PROGRAM P4_01_Write
VAR
	fbDBWrite		:FB_PLCDBWriteEvt(sNetId:=CONST.AMS_NETID, tTimeout:=DEFAULT_ADS_TIMEOUT);

	tableColumns	:ARRAY [0..5] OF STRING(50) := ['DateTime', 'User', 'Event', 'Description', 'OldValue', 'NewValue'];



	
	fbRecipeGeneral				:ARRAY[0..9] OF FB_AuditTrail_Write;
	fbRecipeProduction			:ARRAY[0..49] OF FB_AuditTrail_Write;
	fbRecipeCleaning			:ARRAY[0..49] OF FB_AuditTrail_Write;
	fbBatchProduction			:ARRAY[0..49] OF FB_AuditTrail_Write;
	fbBatchCleaning				:ARRAY[0..49] OF FB_AuditTrail_Write;
	
	fbMachine					:ARRAY[0..49] OF FB_AuditTrail_Write;
	fbSP						:ARRAY[0..49] OF FB_AuditTrail_Write;
	stDBParam 					:ST_AuditTrail;	
	
	//Cmd
	bWrite						:BOOL;								 
	bRead						:BOOL;
	sCmd						:STRING[300];
	nRecords					:UDINT;
	bFilter						:BOOL;
END_VAR

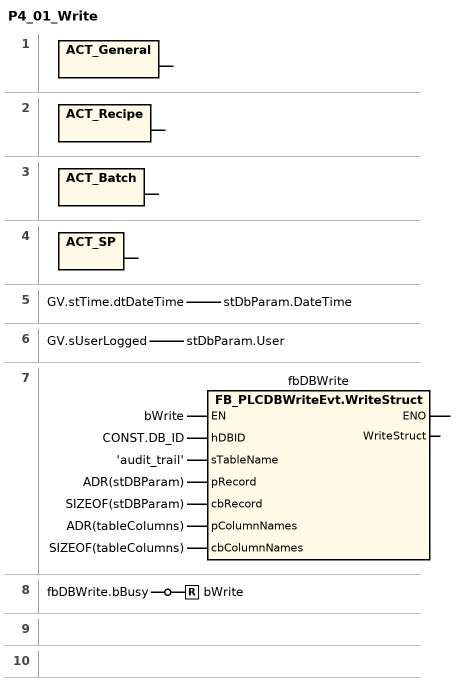
// NETWORK 1
ACT_General();

// NETWORK 2
ACT_Recipe();

// NETWORK 3
ACT_Batch();

// NETWORK 4
ACT_SP();

// NETWORK 5
stDbParam.DateTime := GV.stTime.dtDateTime;

// NETWORK 6
stDbParam.User := GV.sUserLogged;

// NETWORK 7
IF bWrite THEN
    fbDBWrite.WriteStruct(
        hDBID := CONST.DB_ID,
        sTableName := 'audit_trail',
        pRecord := ADR(stDBParam),
        cbRecord := SIZEOF(stDBParam),
        pColumnNames := ADR(tableColumns),
        cbColumnNames := SIZEOF(tableColumns));
END_IF

// NETWORK 8
bWrite R= NOT fbDBWrite.bBusy;

// NETWORK 9

// NETWORK 10

ACTION ACT_Batch:
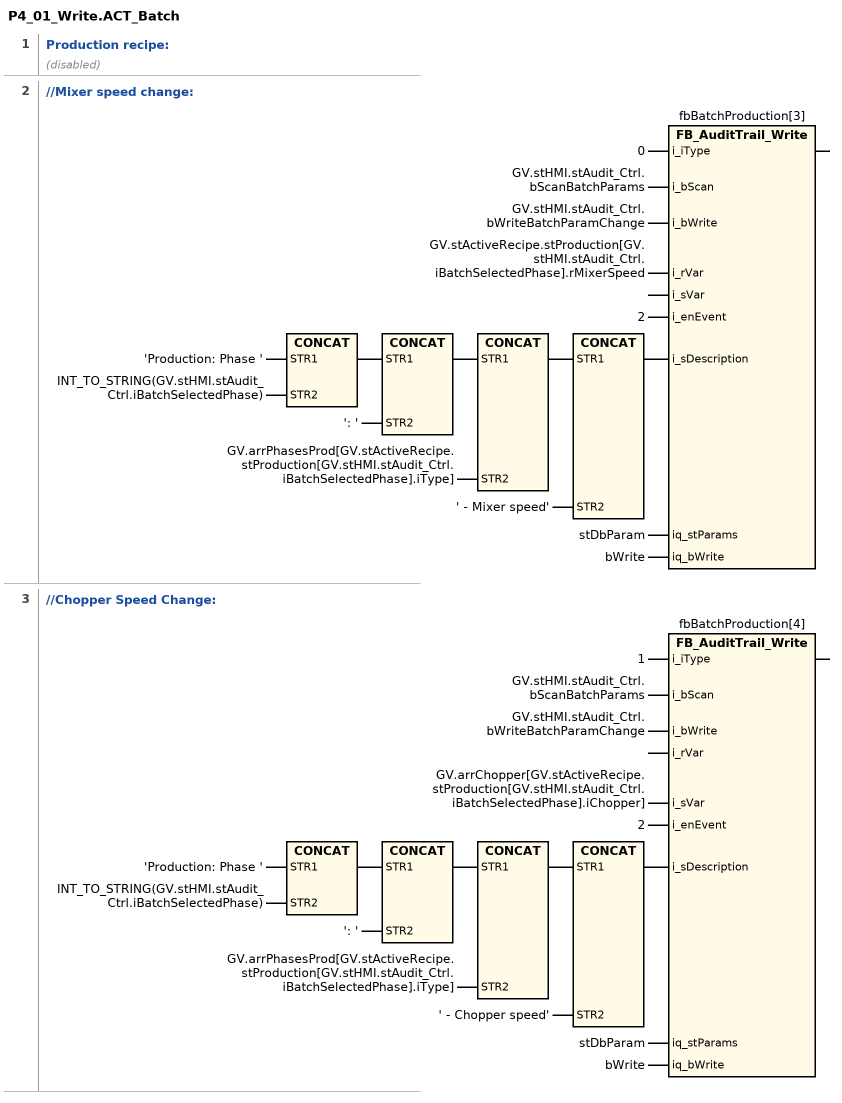
// NETWORK 1 (disabled)
// label: Production recipe

// NETWORK 2
// label: //Mixer speed change
fbBatchProduction[3](
    i_iType := 0,
    i_bScan := GV.stHMI.stAudit_Ctrl.bScanBatchParams,
    i_bWrite := GV.stHMI.stAudit_Ctrl.bWriteBatchParamChange,
    i_rVar := GV.stActiveRecipe.stProduction[GV.stHMI.stAudit_Ctrl.iBatchSelectedPhase].rMixerSpeed,
    i_enEvent := 2,
    i_sDescription := CONCAT(STR1 := CONCAT(STR1 := CONCAT(STR1 := CONCAT(STR1 := 'Production: Phase ', STR2 := INT_TO_STRING(GV.stHMI.stAudit_Ctrl.iBatchSelectedPhase)), STR2 := ': '), STR2 := GV.arrPhasesProd[GV.stActiveRecipe.stProduction[GV.stHMI.stAudit_Ctrl.iBatchSelectedPhase].iType]), STR2 := ' - Mixer speed'),
    iq_stParams := stDbParam,
    iq_bWrite := bWrite); // FB_AuditTrail_Write

// NETWORK 3
// label: //Chopper Speed Change
fbBatchProduction[4](
    i_iType := 1,
    i_bScan := GV.stHMI.stAudit_Ctrl.bScanBatchParams,
    i_bWrite := GV.stHMI.stAudit_Ctrl.bWriteBatchParamChange,
    i_sVar := GV.arrChopper[GV.stActiveRecipe.stProduction[GV.stHMI.stAudit_Ctrl.iBatchSelectedPhase].iChopper],
    i_enEvent := 2,
    i_sDescription := CONCAT(STR1 := CONCAT(STR1 := CONCAT(STR1 := CONCAT(STR1 := 'Production: Phase ', STR2 := INT_TO_STRING(GV.stHMI.stAudit_Ctrl.iBatchSelectedPhase)), STR2 := ': '), STR2 := GV.arrPhasesProd[GV.stActiveRecipe.stProduction[GV.stHMI.stAudit_Ctrl.iBatchSelectedPhase].iType]), STR2 := ' - Chopper speed'),
    iq_stParams := stDbParam,
    iq_bWrite := bWrite); // FB_AuditTrail_Write

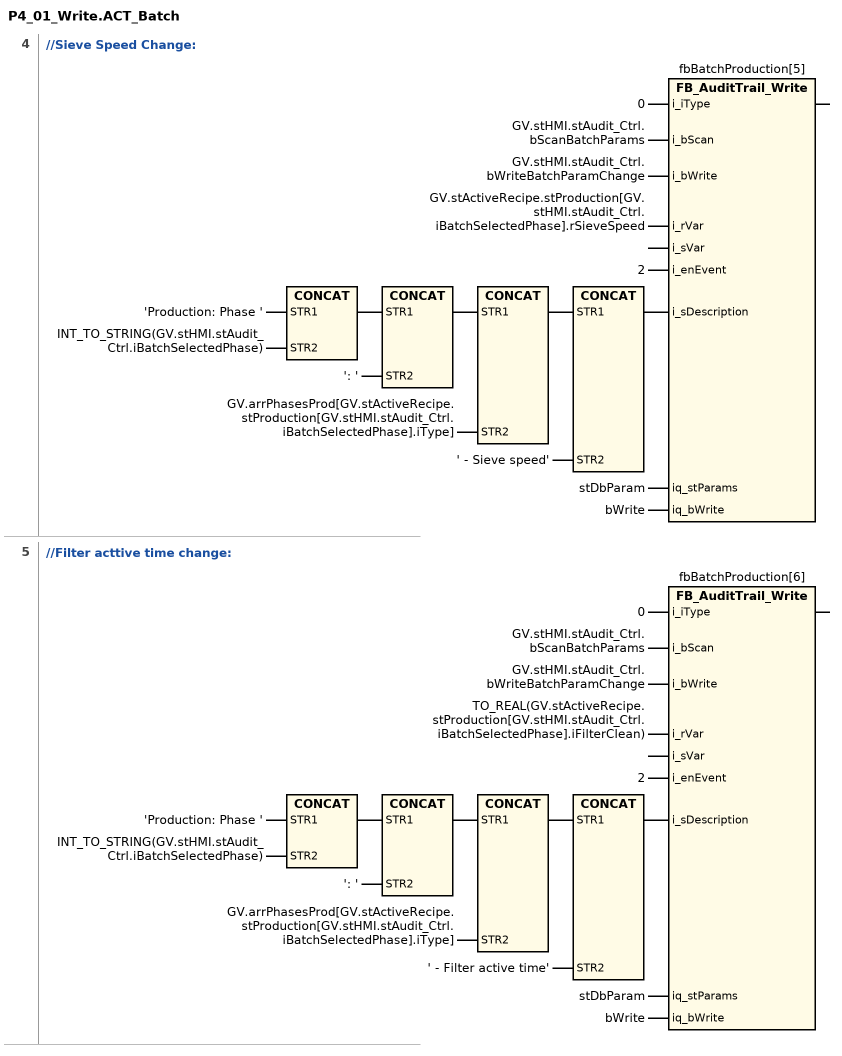
// NETWORK 4
// label: //Sieve Speed Change
fbBatchProduction[5](
    i_iType := 0,
    i_bScan := GV.stHMI.stAudit_Ctrl.bScanBatchParams,
    i_bWrite := GV.stHMI.stAudit_Ctrl.bWriteBatchParamChange,
    i_rVar := GV.stActiveRecipe.stProduction[GV.stHMI.stAudit_Ctrl.iBatchSelectedPhase].rSieveSpeed,
    i_enEvent := 2,
    i_sDescription := CONCAT(STR1 := CONCAT(STR1 := CONCAT(STR1 := CONCAT(STR1 := 'Production: Phase ', STR2 := INT_TO_STRING(GV.stHMI.stAudit_Ctrl.iBatchSelectedPhase)), STR2 := ': '), STR2 := GV.arrPhasesProd[GV.stActiveRecipe.stProduction[GV.stHMI.stAudit_Ctrl.iBatchSelectedPhase].iType]), STR2 := ' - Sieve speed'),
    iq_stParams := stDbParam,
    iq_bWrite := bWrite); // FB_AuditTrail_Write

// NETWORK 5
// label: //Filter acttive time change
fbBatchProduction[6](
    i_iType := 0,
    i_bScan := GV.stHMI.stAudit_Ctrl.bScanBatchParams,
    i_bWrite := GV.stHMI.stAudit_Ctrl.bWriteBatchParamChange,
    i_rVar := TO_REAL(GV.stActiveRecipe.stProduction[GV.stHMI.stAudit_Ctrl.iBatchSelectedPhase].iFilterClean),
    i_enEvent := 2,
    i_sDescription := CONCAT(STR1 := CONCAT(STR1 := CONCAT(STR1 := CONCAT(STR1 := 'Production: Phase ', STR2 := INT_TO_STRING(GV.stHMI.stAudit_Ctrl.iBatchSelectedPhase)), STR2 := ': '), STR2 := GV.arrPhasesProd[GV.stActiveRecipe.stProduction[GV.stHMI.stAudit_Ctrl.iBatchSelectedPhase].iType]), STR2 := ' - Filter active time'),
    iq_stParams := stDbParam,
    iq_bWrite := bWrite); // FB_AuditTrail_Write

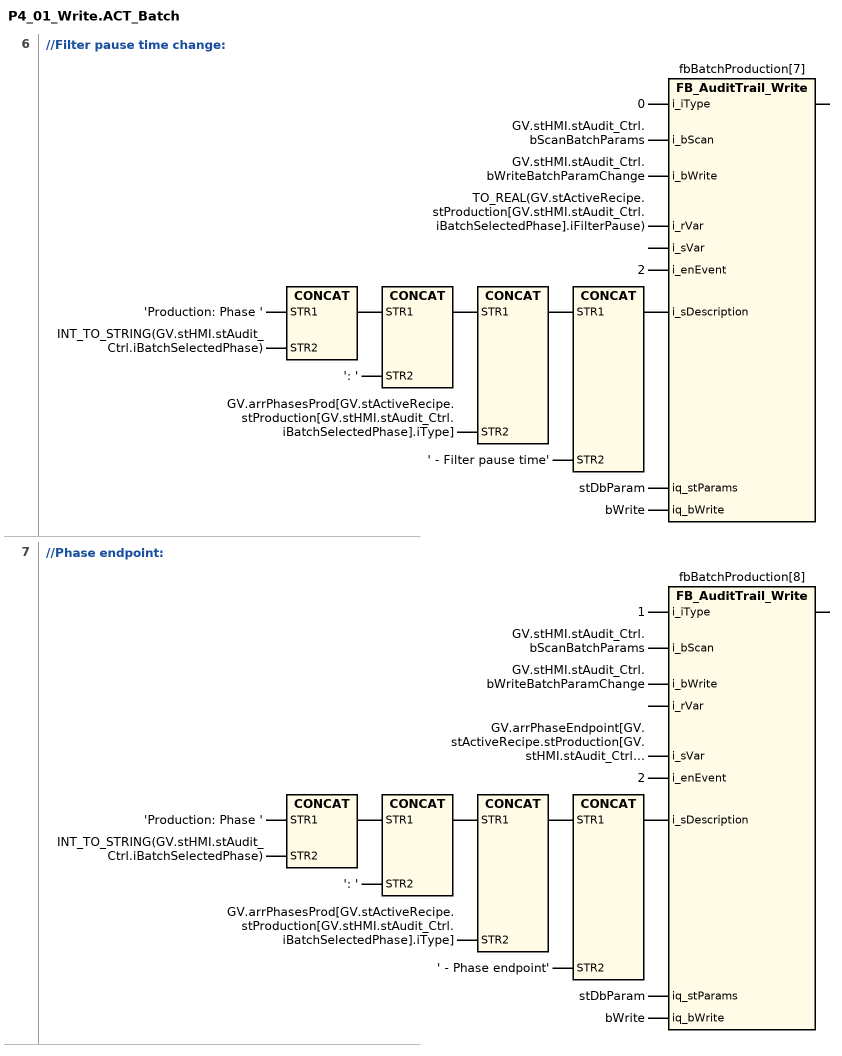
// NETWORK 6
// label: //Filter pause time change
fbBatchProduction[7](
    i_iType := 0,
    i_bScan := GV.stHMI.stAudit_Ctrl.bScanBatchParams,
    i_bWrite := GV.stHMI.stAudit_Ctrl.bWriteBatchParamChange,
    i_rVar := TO_REAL(GV.stActiveRecipe.stProduction[GV.stHMI.stAudit_Ctrl.iBatchSelectedPhase].iFilterPause),
    i_enEvent := 2,
    i_sDescription := CONCAT(STR1 := CONCAT(STR1 := CONCAT(STR1 := CONCAT(STR1 := 'Production: Phase ', STR2 := INT_TO_STRING(GV.stHMI.stAudit_Ctrl.iBatchSelectedPhase)), STR2 := ': '), STR2 := GV.arrPhasesProd[GV.stActiveRecipe.stProduction[GV.stHMI.stAudit_Ctrl.iBatchSelectedPhase].iType]), STR2 := ' - Filter pause time'),
    iq_stParams := stDbParam,
    iq_bWrite := bWrite); // FB_AuditTrail_Write

// NETWORK 7
// label: //Phase endpoint
fbBatchProduction[8](
    i_iType := 1,
    i_bScan := GV.stHMI.stAudit_Ctrl.bScanBatchParams,
    i_bWrite := GV.stHMI.stAudit_Ctrl.bWriteBatchParamChange,
    i_sVar := GV.arrPhaseEndpoint[GV.stActiveRecipe.stProduction[GV.stHMI.stAudit_Ctrl.iBatchSelectedPhase].iEndPoint],
    i_enEvent := 2,
    i_sDescription := CONCAT(STR1 := CONCAT(STR1 := CONCAT(STR1 := CONCAT(STR1 := 'Production: Phase ', STR2 := INT_TO_STRING(GV.stHMI.stAudit_Ctrl.iBatchSelectedPhase)), STR2 := ': '), STR2 := GV.arrPhasesProd[GV.stActiveRecipe.stProduction[GV.stHMI.stAudit_Ctrl.iBatchSelectedPhase].iType]), STR2 := ' - Phase endpoint'),
    iq_stParams := stDbParam,
    iq_bWrite := bWrite); // FB_AuditTrail_Write

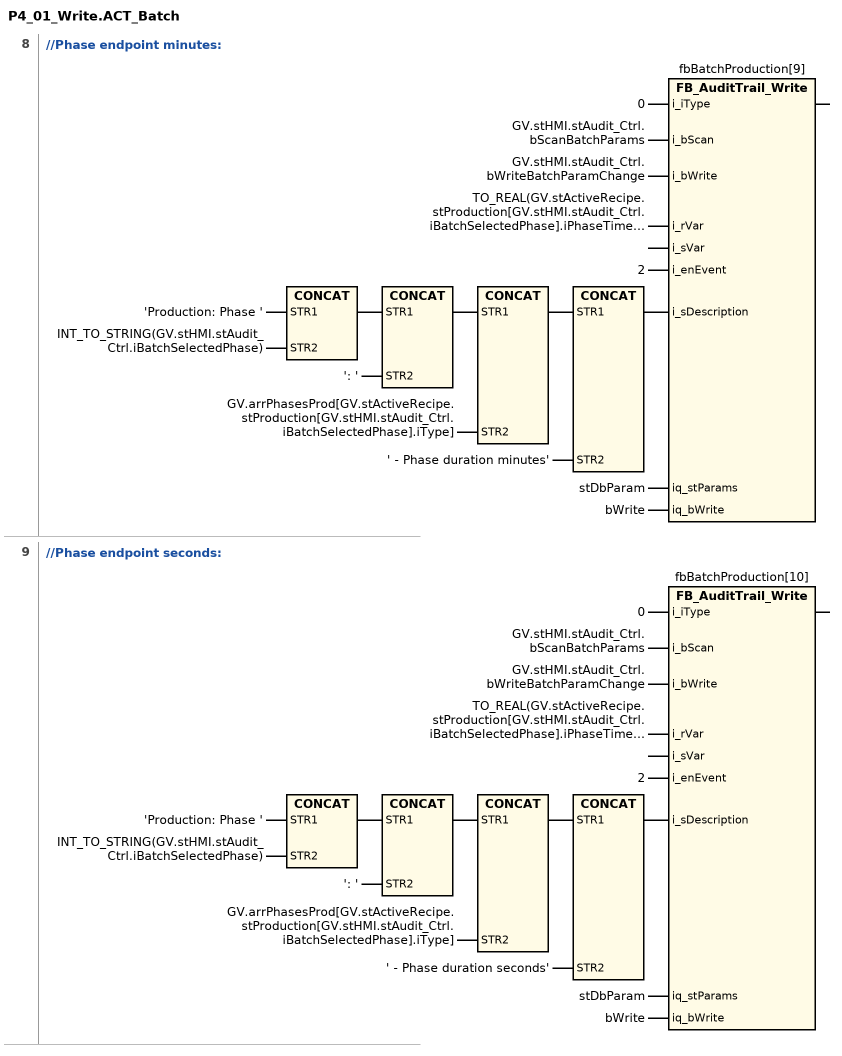
// NETWORK 8
// label: //Phase endpoint minutes
fbBatchProduction[9](
    i_iType := 0,
    i_bScan := GV.stHMI.stAudit_Ctrl.bScanBatchParams,
    i_bWrite := GV.stHMI.stAudit_Ctrl.bWriteBatchParamChange,
    i_rVar := TO_REAL(GV.stActiveRecipe.stProduction[GV.stHMI.stAudit_Ctrl.iBatchSelectedPhase].iPhaseTime.mins),
    i_enEvent := 2,
    i_sDescription := CONCAT(STR1 := CONCAT(STR1 := CONCAT(STR1 := CONCAT(STR1 := 'Production: Phase ', STR2 := INT_TO_STRING(GV.stHMI.stAudit_Ctrl.iBatchSelectedPhase)), STR2 := ': '), STR2 := GV.arrPhasesProd[GV.stActiveRecipe.stProduction[GV.stHMI.stAudit_Ctrl.iBatchSelectedPhase].iType]), STR2 := ' - Phase duration minutes'),
    iq_stParams := stDbParam,
    iq_bWrite := bWrite); // FB_AuditTrail_Write

// NETWORK 9
// label: //Phase endpoint seconds
fbBatchProduction[10](
    i_iType := 0,
    i_bScan := GV.stHMI.stAudit_Ctrl.bScanBatchParams,
    i_bWrite := GV.stHMI.stAudit_Ctrl.bWriteBatchParamChange,
    i_rVar := TO_REAL(GV.stActiveRecipe.stProduction[GV.stHMI.stAudit_Ctrl.iBatchSelectedPhase].iPhaseTime.sec),
    i_enEvent := 2,
    i_sDescription := CONCAT(STR1 := CONCAT(STR1 := CONCAT(STR1 := CONCAT(STR1 := 'Production: Phase ', STR2 := INT_TO_STRING(GV.stHMI.stAudit_Ctrl.iBatchSelectedPhase)), STR2 := ': '), STR2 := GV.arrPhasesProd[GV.stActiveRecipe.stProduction[GV.stHMI.stAudit_Ctrl.iBatchSelectedPhase].iType]), STR2 := ' - Phase duration seconds'),
    iq_stParams := stDbParam,
    iq_bWrite := bWrite); // FB_AuditTrail_Write

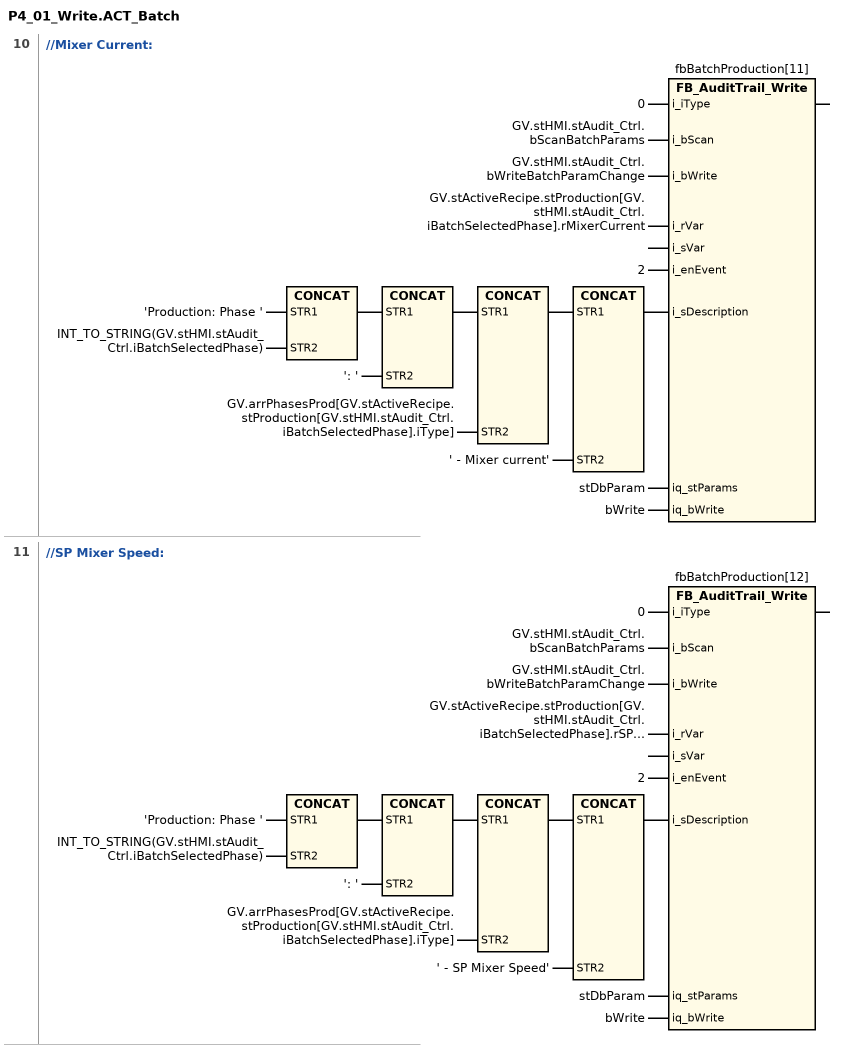
// NETWORK 10
// label: //Mixer Current
fbBatchProduction[11](
    i_iType := 0,
    i_bScan := GV.stHMI.stAudit_Ctrl.bScanBatchParams,
    i_bWrite := GV.stHMI.stAudit_Ctrl.bWriteBatchParamChange,
    i_rVar := GV.stActiveRecipe.stProduction[GV.stHMI.stAudit_Ctrl.iBatchSelectedPhase].rMixerCurrent,
    i_enEvent := 2,
    i_sDescription := CONCAT(STR1 := CONCAT(STR1 := CONCAT(STR1 := CONCAT(STR1 := 'Production: Phase ', STR2 := INT_TO_STRING(GV.stHMI.stAudit_Ctrl.iBatchSelectedPhase)), STR2 := ': '), STR2 := GV.arrPhasesProd[GV.stActiveRecipe.stProduction[GV.stHMI.stAudit_Ctrl.iBatchSelectedPhase].iType]), STR2 := ' - Mixer current'),
    iq_stParams := stDbParam,
    iq_bWrite := bWrite); // FB_AuditTrail_Write

// NETWORK 11
// label: //SP Mixer Speed
fbBatchProduction[12](
    i_iType := 0,
    i_bScan := GV.stHMI.stAudit_Ctrl.bScanBatchParams,
    i_bWrite := GV.stHMI.stAudit_Ctrl.bWriteBatchParamChange,
    i_rVar := GV.stActiveRecipe.stProduction[GV.stHMI.stAudit_Ctrl.iBatchSelectedPhase].rSP_MixingSpeed,
    i_enEvent := 2,
    i_sDescription := CONCAT(STR1 := CONCAT(STR1 := CONCAT(STR1 := CONCAT(STR1 := 'Production: Phase ', STR2 := INT_TO_STRING(GV.stHMI.stAudit_Ctrl.iBatchSelectedPhase)), STR2 := ': '), STR2 := GV.arrPhasesProd[GV.stActiveRecipe.stProduction[GV.stHMI.stAudit_Ctrl.iBatchSelectedPhase].iType]), STR2 := ' - SP Mixer Speed'),
    iq_stParams := stDbParam,
    iq_bWrite := bWrite); // FB_AuditTrail_Write

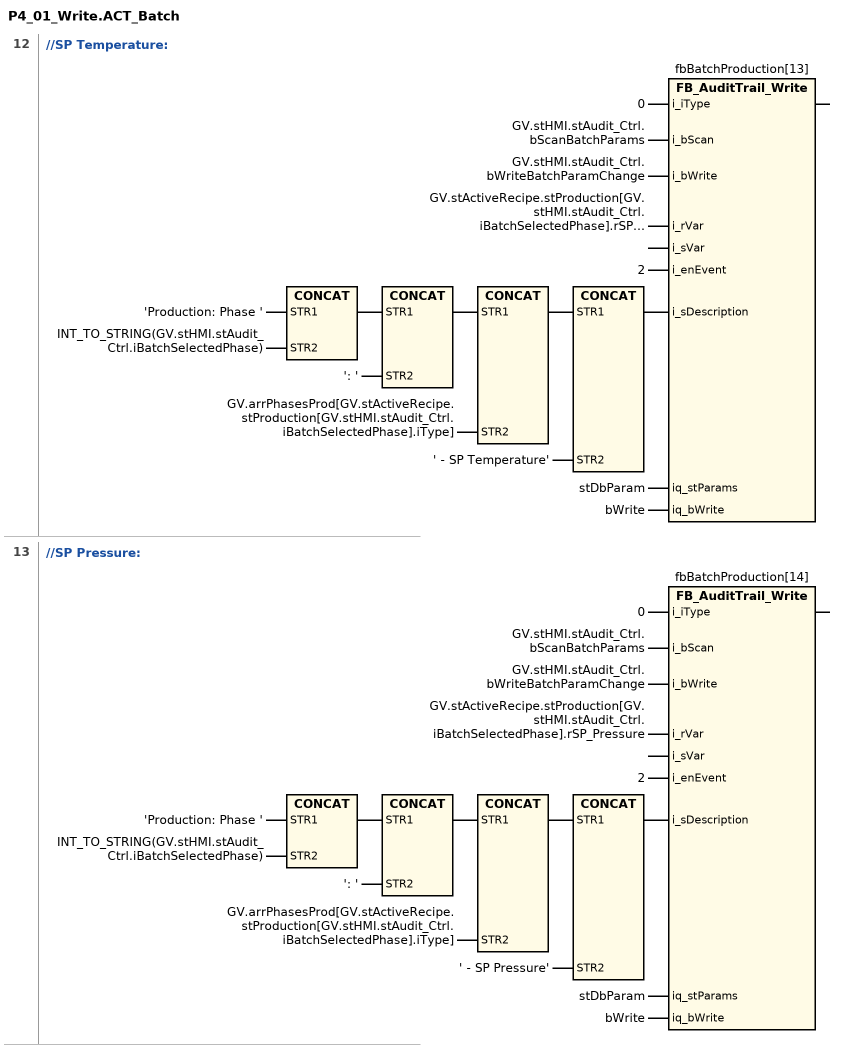
// NETWORK 12
// label: //SP Temperature
fbBatchProduction[13](
    i_iType := 0,
    i_bScan := GV.stHMI.stAudit_Ctrl.bScanBatchParams,
    i_bWrite := GV.stHMI.stAudit_Ctrl.bWriteBatchParamChange,
    i_rVar := GV.stActiveRecipe.stProduction[GV.stHMI.stAudit_Ctrl.iBatchSelectedPhase].rSP_Temperature,
    i_enEvent := 2,
    i_sDescription := CONCAT(STR1 := CONCAT(STR1 := CONCAT(STR1 := CONCAT(STR1 := 'Production: Phase ', STR2 := INT_TO_STRING(GV.stHMI.stAudit_Ctrl.iBatchSelectedPhase)), STR2 := ': '), STR2 := GV.arrPhasesProd[GV.stActiveRecipe.stProduction[GV.stHMI.stAudit_Ctrl.iBatchSelectedPhase].iType]), STR2 := ' - SP Temperature'),
    iq_stParams := stDbParam,
    iq_bWrite := bWrite); // FB_AuditTrail_Write

// NETWORK 13
// label: //SP Pressure
fbBatchProduction[14](
    i_iType := 0,
    i_bScan := GV.stHMI.stAudit_Ctrl.bScanBatchParams,
    i_bWrite := GV.stHMI.stAudit_Ctrl.bWriteBatchParamChange,
    i_rVar := GV.stActiveRecipe.stProduction[GV.stHMI.stAudit_Ctrl.iBatchSelectedPhase].rSP_Pressure,
    i_enEvent := 2,
    i_sDescription := CONCAT(STR1 := CONCAT(STR1 := CONCAT(STR1 := CONCAT(STR1 := 'Production: Phase ', STR2 := INT_TO_STRING(GV.stHMI.stAudit_Ctrl.iBatchSelectedPhase)), STR2 := ': '), STR2 := GV.arrPhasesProd[GV.stActiveRecipe.stProduction[GV.stHMI.stAudit_Ctrl.iBatchSelectedPhase].iType]), STR2 := ' - SP Pressure'),
    iq_stParams := stDbParam,
    iq_bWrite := bWrite); // FB_AuditTrail_Write

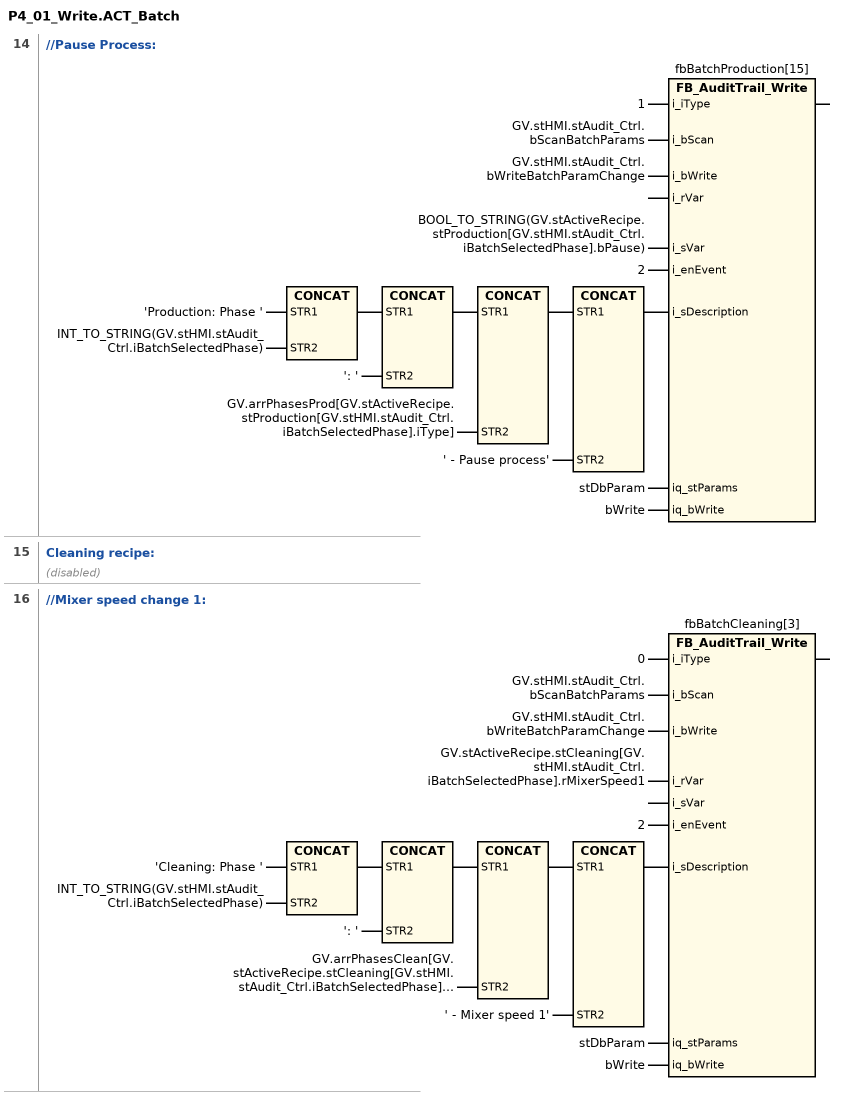
// NETWORK 14
// label: //Pause Process
fbBatchProduction[15](
    i_iType := 1,
    i_bScan := GV.stHMI.stAudit_Ctrl.bScanBatchParams,
    i_bWrite := GV.stHMI.stAudit_Ctrl.bWriteBatchParamChange,
    i_sVar := BOOL_TO_STRING(GV.stActiveRecipe.stProduction[GV.stHMI.stAudit_Ctrl.iBatchSelectedPhase].bPause),
    i_enEvent := 2,
    i_sDescription := CONCAT(STR1 := CONCAT(STR1 := CONCAT(STR1 := CONCAT(STR1 := 'Production: Phase ', STR2 := INT_TO_STRING(GV.stHMI.stAudit_Ctrl.iBatchSelectedPhase)), STR2 := ': '), STR2 := GV.arrPhasesProd[GV.stActiveRecipe.stProduction[GV.stHMI.stAudit_Ctrl.iBatchSelectedPhase].iType]), STR2 := ' - Pause process'),
    iq_stParams := stDbParam,
    iq_bWrite := bWrite); // FB_AuditTrail_Write

// NETWORK 15 (disabled)
// label: Cleaning recipe

// NETWORK 16
// label: //Mixer speed change 1
fbBatchCleaning[3](
    i_iType := 0,
    i_bScan := GV.stHMI.stAudit_Ctrl.bScanBatchParams,
    i_bWrite := GV.stHMI.stAudit_Ctrl.bWriteBatchParamChange,
    i_rVar := GV.stActiveRecipe.stCleaning[GV.stHMI.stAudit_Ctrl.iBatchSelectedPhase].rMixerSpeed1,
    i_enEvent := 2,
    i_sDescription := CONCAT(STR1 := CONCAT(STR1 := CONCAT(STR1 := CONCAT(STR1 := 'Cleaning: Phase ', STR2 := INT_TO_STRING(GV.stHMI.stAudit_Ctrl.iBatchSelectedPhase)), STR2 := ': '), STR2 := GV.arrPhasesClean[GV.stActiveRecipe.stCleaning[GV.stHMI.stAudit_Ctrl.iBatchSelectedPhase].iType]), STR2 := ' - Mixer speed 1'),
    iq_stParams := stDbParam,
    iq_bWrite := bWrite); // FB_AuditTrail_Write

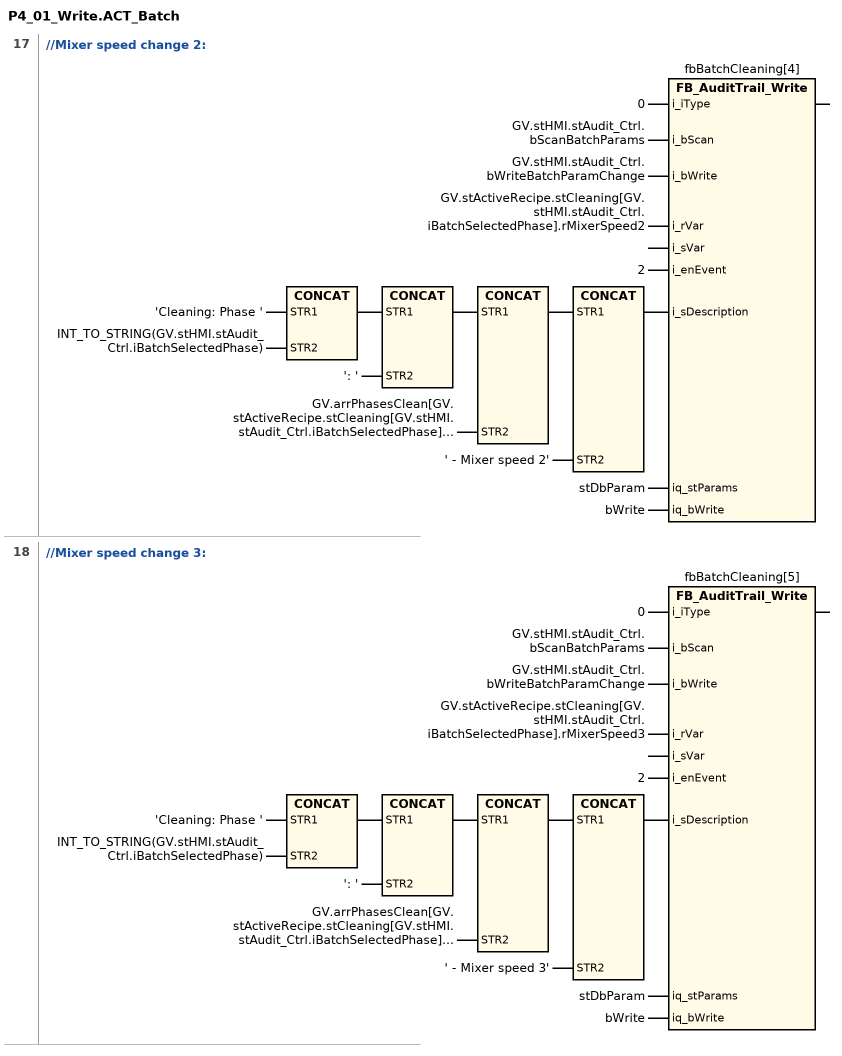
// NETWORK 17
// label: //Mixer speed change 2
fbBatchCleaning[4](
    i_iType := 0,
    i_bScan := GV.stHMI.stAudit_Ctrl.bScanBatchParams,
    i_bWrite := GV.stHMI.stAudit_Ctrl.bWriteBatchParamChange,
    i_rVar := GV.stActiveRecipe.stCleaning[GV.stHMI.stAudit_Ctrl.iBatchSelectedPhase].rMixerSpeed2,
    i_enEvent := 2,
    i_sDescription := CONCAT(STR1 := CONCAT(STR1 := CONCAT(STR1 := CONCAT(STR1 := 'Cleaning: Phase ', STR2 := INT_TO_STRING(GV.stHMI.stAudit_Ctrl.iBatchSelectedPhase)), STR2 := ': '), STR2 := GV.arrPhasesClean[GV.stActiveRecipe.stCleaning[GV.stHMI.stAudit_Ctrl.iBatchSelectedPhase].iType]), STR2 := ' - Mixer speed 2'),
    iq_stParams := stDbParam,
    iq_bWrite := bWrite); // FB_AuditTrail_Write

// NETWORK 18
// label: //Mixer speed change 3
fbBatchCleaning[5](
    i_iType := 0,
    i_bScan := GV.stHMI.stAudit_Ctrl.bScanBatchParams,
    i_bWrite := GV.stHMI.stAudit_Ctrl.bWriteBatchParamChange,
    i_rVar := GV.stActiveRecipe.stCleaning[GV.stHMI.stAudit_Ctrl.iBatchSelectedPhase].rMixerSpeed3,
    i_enEvent := 2,
    i_sDescription := CONCAT(STR1 := CONCAT(STR1 := CONCAT(STR1 := CONCAT(STR1 := 'Cleaning: Phase ', STR2 := INT_TO_STRING(GV.stHMI.stAudit_Ctrl.iBatchSelectedPhase)), STR2 := ': '), STR2 := GV.arrPhasesClean[GV.stActiveRecipe.stCleaning[GV.stHMI.stAudit_Ctrl.iBatchSelectedPhase].iType]), STR2 := ' - Mixer speed 3'),
    iq_stParams := stDbParam,
    iq_bWrite := bWrite); // FB_AuditTrail_Write

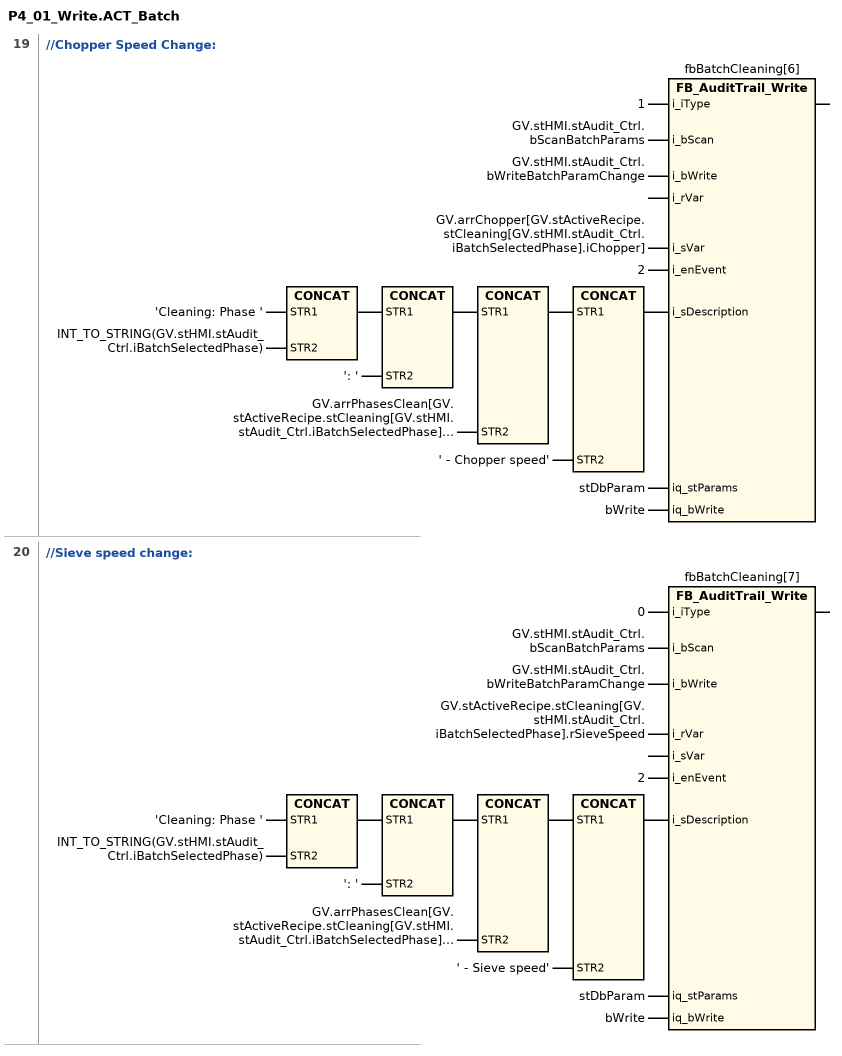
// NETWORK 19
// label: //Chopper Speed Change
fbBatchCleaning[6](
    i_iType := 1,
    i_bScan := GV.stHMI.stAudit_Ctrl.bScanBatchParams,
    i_bWrite := GV.stHMI.stAudit_Ctrl.bWriteBatchParamChange,
    i_sVar := GV.arrChopper[GV.stActiveRecipe.stCleaning[GV.stHMI.stAudit_Ctrl.iBatchSelectedPhase].iChopper],
    i_enEvent := 2,
    i_sDescription := CONCAT(STR1 := CONCAT(STR1 := CONCAT(STR1 := CONCAT(STR1 := 'Cleaning: Phase ', STR2 := INT_TO_STRING(GV.stHMI.stAudit_Ctrl.iBatchSelectedPhase)), STR2 := ': '), STR2 := GV.arrPhasesClean[GV.stActiveRecipe.stCleaning[GV.stHMI.stAudit_Ctrl.iBatchSelectedPhase].iType]), STR2 := ' - Chopper speed'),
    iq_stParams := stDbParam,
    iq_bWrite := bWrite); // FB_AuditTrail_Write

// NETWORK 20
// label: //Sieve speed change
fbBatchCleaning[7](
    i_iType := 0,
    i_bScan := GV.stHMI.stAudit_Ctrl.bScanBatchParams,
    i_bWrite := GV.stHMI.stAudit_Ctrl.bWriteBatchParamChange,
    i_rVar := GV.stActiveRecipe.stCleaning[GV.stHMI.stAudit_Ctrl.iBatchSelectedPhase].rSieveSpeed,
    i_enEvent := 2,
    i_sDescription := CONCAT(STR1 := CONCAT(STR1 := CONCAT(STR1 := CONCAT(STR1 := 'Cleaning: Phase ', STR2 := INT_TO_STRING(GV.stHMI.stAudit_Ctrl.iBatchSelectedPhase)), STR2 := ': '), STR2 := GV.arrPhasesClean[GV.stActiveRecipe.stCleaning[GV.stHMI.stAudit_Ctrl.iBatchSelectedPhase].iType]), STR2 := ' - Sieve speed'),
    iq_stParams := stDbParam,
    iq_bWrite := bWrite); // FB_AuditTrail_Write

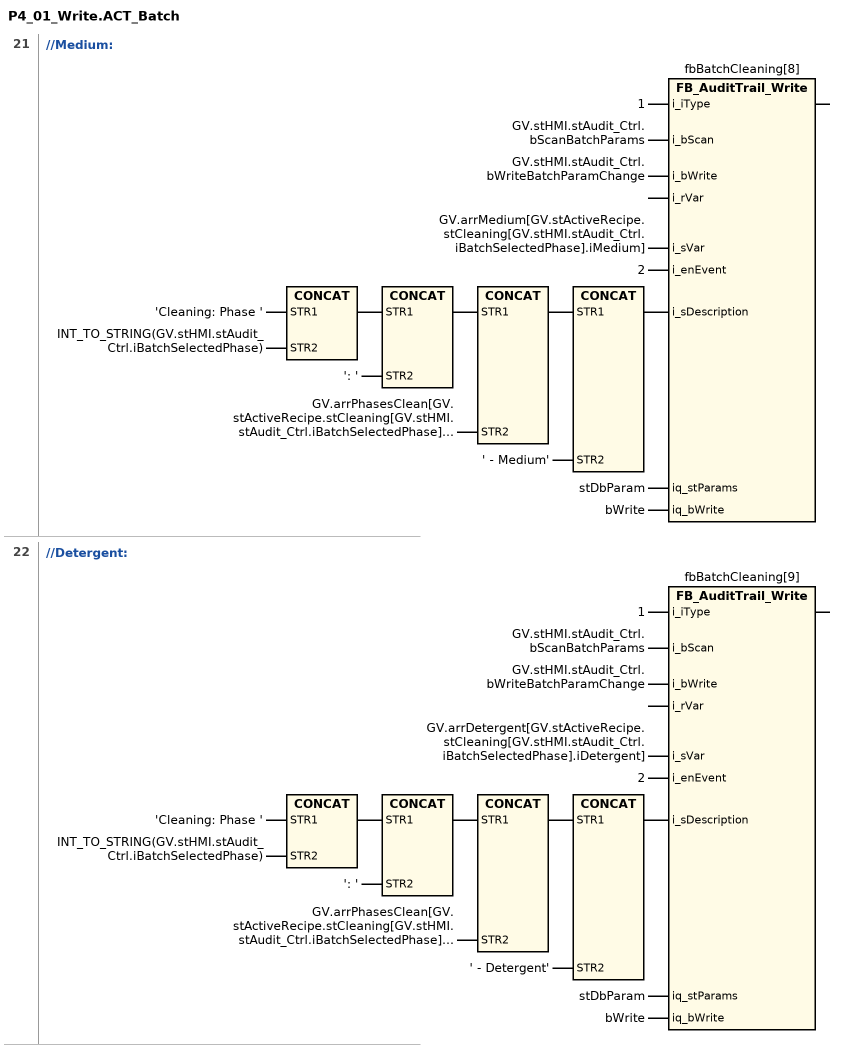
// NETWORK 21
// label: //Medium
fbBatchCleaning[8](
    i_iType := 1,
    i_bScan := GV.stHMI.stAudit_Ctrl.bScanBatchParams,
    i_bWrite := GV.stHMI.stAudit_Ctrl.bWriteBatchParamChange,
    i_sVar := GV.arrMedium[GV.stActiveRecipe.stCleaning[GV.stHMI.stAudit_Ctrl.iBatchSelectedPhase].iMedium],
    i_enEvent := 2,
    i_sDescription := CONCAT(STR1 := CONCAT(STR1 := CONCAT(STR1 := CONCAT(STR1 := 'Cleaning: Phase ', STR2 := INT_TO_STRING(GV.stHMI.stAudit_Ctrl.iBatchSelectedPhase)), STR2 := ': '), STR2 := GV.arrPhasesClean[GV.stActiveRecipe.stCleaning[GV.stHMI.stAudit_Ctrl.iBatchSelectedPhase].iType]), STR2 := ' - Medium'),
    iq_stParams := stDbParam,
    iq_bWrite := bWrite); // FB_AuditTrail_Write

// NETWORK 22
// label: //Detergent
fbBatchCleaning[9](
    i_iType := 1,
    i_bScan := GV.stHMI.stAudit_Ctrl.bScanBatchParams,
    i_bWrite := GV.stHMI.stAudit_Ctrl.bWriteBatchParamChange,
    i_sVar := GV.arrDetergent[GV.stActiveRecipe.stCleaning[GV.stHMI.stAudit_Ctrl.iBatchSelectedPhase].iDetergent],
    i_enEvent := 2,
    i_sDescription := CONCAT(STR1 := CONCAT(STR1 := CONCAT(STR1 := CONCAT(STR1 := 'Cleaning: Phase ', STR2 := INT_TO_STRING(GV.stHMI.stAudit_Ctrl.iBatchSelectedPhase)), STR2 := ': '), STR2 := GV.arrPhasesClean[GV.stActiveRecipe.stCleaning[GV.stHMI.stAudit_Ctrl.iBatchSelectedPhase].iType]), STR2 := ' - Detergent'),
    iq_stParams := stDbParam,
    iq_bWrite := bWrite); // FB_AuditTrail_Write

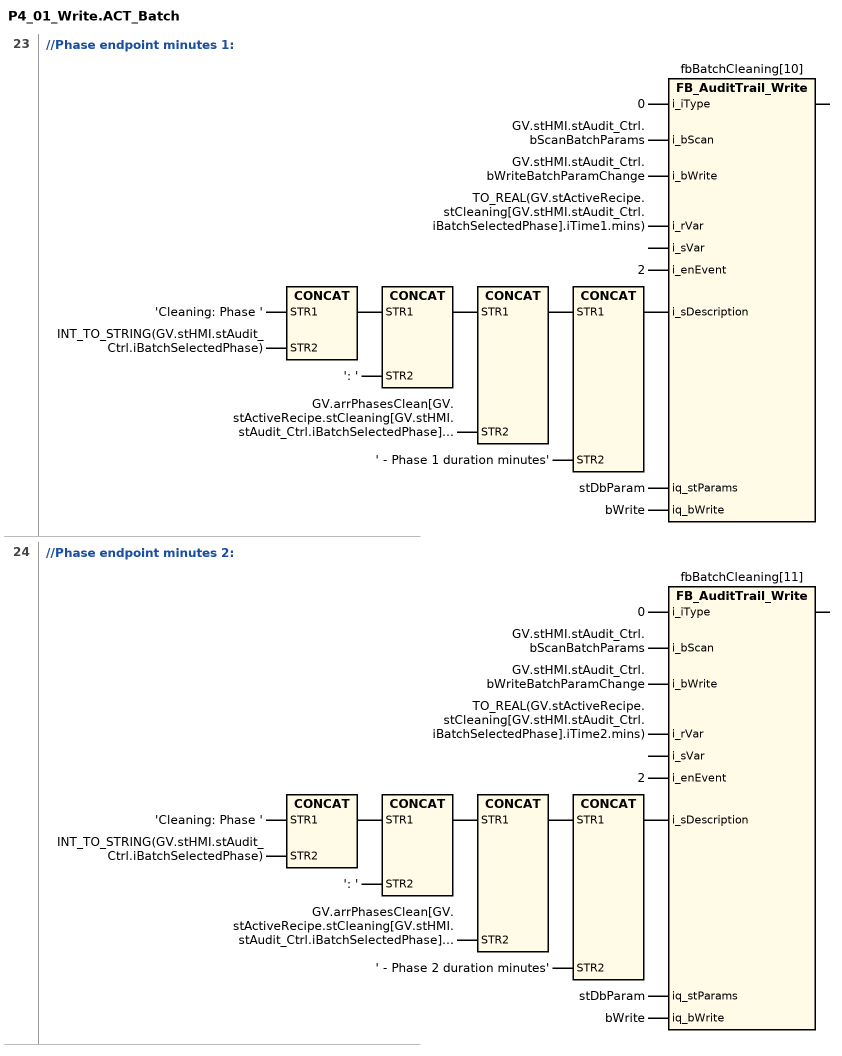
// NETWORK 23
// label: //Phase endpoint minutes 1
fbBatchCleaning[10](
    i_iType := 0,
    i_bScan := GV.stHMI.stAudit_Ctrl.bScanBatchParams,
    i_bWrite := GV.stHMI.stAudit_Ctrl.bWriteBatchParamChange,
    i_rVar := TO_REAL(GV.stActiveRecipe.stCleaning[GV.stHMI.stAudit_Ctrl.iBatchSelectedPhase].iTime1.mins),
    i_enEvent := 2,
    i_sDescription := CONCAT(STR1 := CONCAT(STR1 := CONCAT(STR1 := CONCAT(STR1 := 'Cleaning: Phase ', STR2 := INT_TO_STRING(GV.stHMI.stAudit_Ctrl.iBatchSelectedPhase)), STR2 := ': '), STR2 := GV.arrPhasesClean[GV.stActiveRecipe.stCleaning[GV.stHMI.stAudit_Ctrl.iBatchSelectedPhase].iType]), STR2 := ' - Phase 1 duration minutes'),
    iq_stParams := stDbParam,
    iq_bWrite := bWrite); // FB_AuditTrail_Write

// NETWORK 24
// label: //Phase endpoint minutes 2
fbBatchCleaning[11](
    i_iType := 0,
    i_bScan := GV.stHMI.stAudit_Ctrl.bScanBatchParams,
    i_bWrite := GV.stHMI.stAudit_Ctrl.bWriteBatchParamChange,
    i_rVar := TO_REAL(GV.stActiveRecipe.stCleaning[GV.stHMI.stAudit_Ctrl.iBatchSelectedPhase].iTime2.mins),
    i_enEvent := 2,
    i_sDescription := CONCAT(STR1 := CONCAT(STR1 := CONCAT(STR1 := CONCAT(STR1 := 'Cleaning: Phase ', STR2 := INT_TO_STRING(GV.stHMI.stAudit_Ctrl.iBatchSelectedPhase)), STR2 := ': '), STR2 := GV.arrPhasesClean[GV.stActiveRecipe.stCleaning[GV.stHMI.stAudit_Ctrl.iBatchSelectedPhase].iType]), STR2 := ' - Phase 2 duration minutes'),
    iq_stParams := stDbParam,
    iq_bWrite := bWrite); // FB_AuditTrail_Write

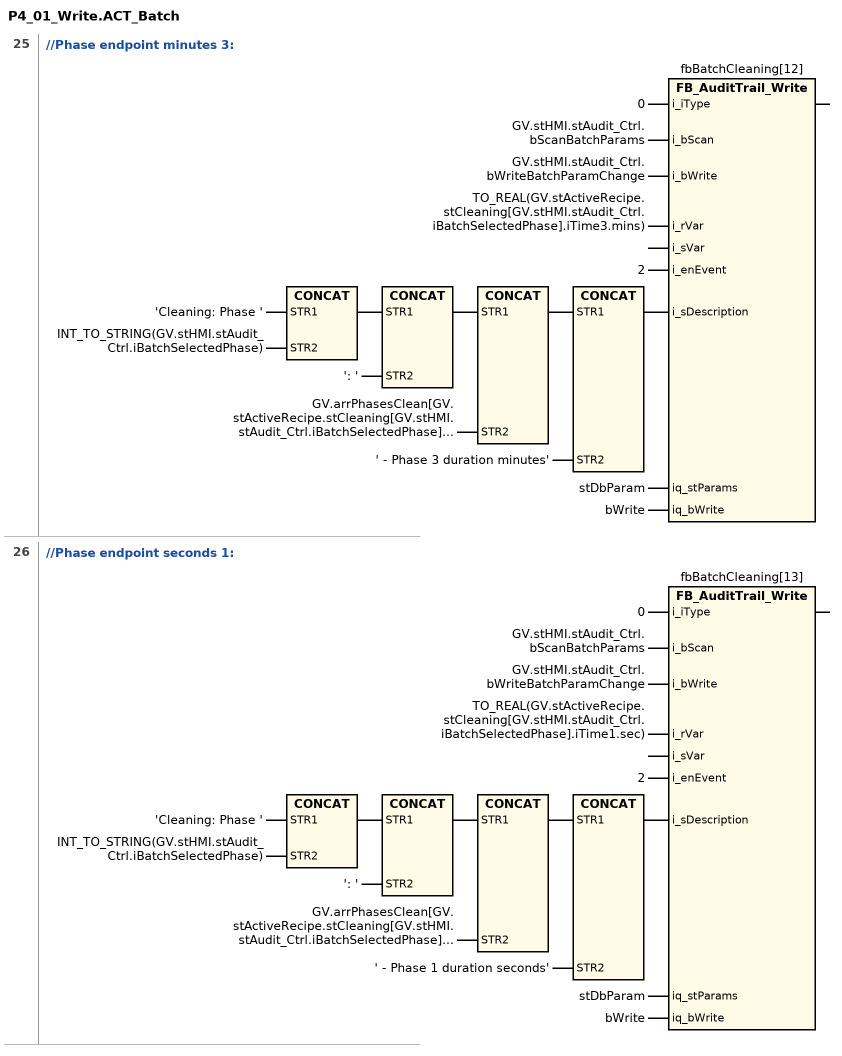
// NETWORK 25
// label: //Phase endpoint minutes 3
fbBatchCleaning[12](
    i_iType := 0,
    i_bScan := GV.stHMI.stAudit_Ctrl.bScanBatchParams,
    i_bWrite := GV.stHMI.stAudit_Ctrl.bWriteBatchParamChange,
    i_rVar := TO_REAL(GV.stActiveRecipe.stCleaning[GV.stHMI.stAudit_Ctrl.iBatchSelectedPhase].iTime3.mins),
    i_enEvent := 2,
    i_sDescription := CONCAT(STR1 := CONCAT(STR1 := CONCAT(STR1 := CONCAT(STR1 := 'Cleaning: Phase ', STR2 := INT_TO_STRING(GV.stHMI.stAudit_Ctrl.iBatchSelectedPhase)), STR2 := ': '), STR2 := GV.arrPhasesClean[GV.stActiveRecipe.stCleaning[GV.stHMI.stAudit_Ctrl.iBatchSelectedPhase].iType]), STR2 := ' - Phase 3 duration minutes'),
    iq_stParams := stDbParam,
    iq_bWrite := bWrite); // FB_AuditTrail_Write

// NETWORK 26
// label: //Phase endpoint seconds 1
fbBatchCleaning[13](
    i_iType := 0,
    i_bScan := GV.stHMI.stAudit_Ctrl.bScanBatchParams,
    i_bWrite := GV.stHMI.stAudit_Ctrl.bWriteBatchParamChange,
    i_rVar := TO_REAL(GV.stActiveRecipe.stCleaning[GV.stHMI.stAudit_Ctrl.iBatchSelectedPhase].iTime1.sec),
    i_enEvent := 2,
    i_sDescription := CONCAT(STR1 := CONCAT(STR1 := CONCAT(STR1 := CONCAT(STR1 := 'Cleaning: Phase ', STR2 := INT_TO_STRING(GV.stHMI.stAudit_Ctrl.iBatchSelectedPhase)), STR2 := ': '), STR2 := GV.arrPhasesClean[GV.stActiveRecipe.stCleaning[GV.stHMI.stAudit_Ctrl.iBatchSelectedPhase].iType]), STR2 := ' - Phase 1 duration seconds'),
    iq_stParams := stDbParam,
    iq_bWrite := bWrite); // FB_AuditTrail_Write

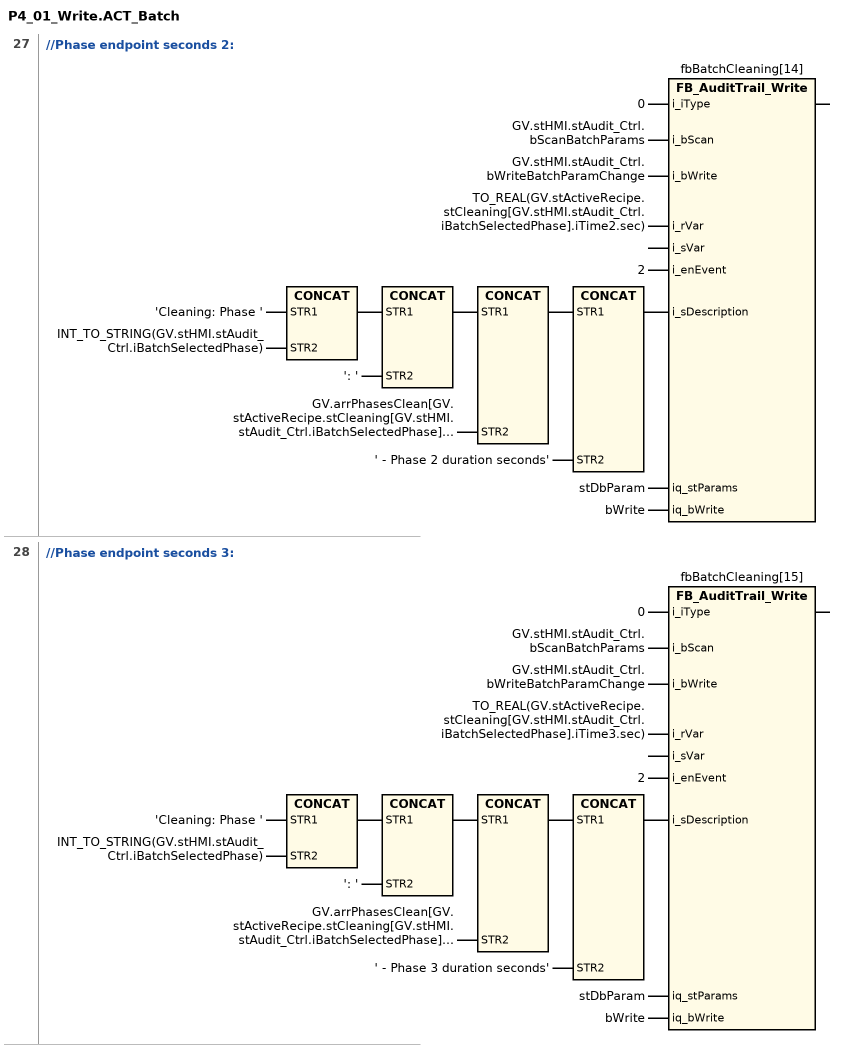
// NETWORK 27
// label: //Phase endpoint seconds 2
fbBatchCleaning[14](
    i_iType := 0,
    i_bScan := GV.stHMI.stAudit_Ctrl.bScanBatchParams,
    i_bWrite := GV.stHMI.stAudit_Ctrl.bWriteBatchParamChange,
    i_rVar := TO_REAL(GV.stActiveRecipe.stCleaning[GV.stHMI.stAudit_Ctrl.iBatchSelectedPhase].iTime2.sec),
    i_enEvent := 2,
    i_sDescription := CONCAT(STR1 := CONCAT(STR1 := CONCAT(STR1 := CONCAT(STR1 := 'Cleaning: Phase ', STR2 := INT_TO_STRING(GV.stHMI.stAudit_Ctrl.iBatchSelectedPhase)), STR2 := ': '), STR2 := GV.arrPhasesClean[GV.stActiveRecipe.stCleaning[GV.stHMI.stAudit_Ctrl.iBatchSelectedPhase].iType]), STR2 := ' - Phase 2 duration seconds'),
    iq_stParams := stDbParam,
    iq_bWrite := bWrite); // FB_AuditTrail_Write

// NETWORK 28
// label: //Phase endpoint seconds 3
fbBatchCleaning[15](
    i_iType := 0,
    i_bScan := GV.stHMI.stAudit_Ctrl.bScanBatchParams,
    i_bWrite := GV.stHMI.stAudit_Ctrl.bWriteBatchParamChange,
    i_rVar := TO_REAL(GV.stActiveRecipe.stCleaning[GV.stHMI.stAudit_Ctrl.iBatchSelectedPhase].iTime3.sec),
    i_enEvent := 2,
    i_sDescription := CONCAT(STR1 := CONCAT(STR1 := CONCAT(STR1 := CONCAT(STR1 := 'Cleaning: Phase ', STR2 := INT_TO_STRING(GV.stHMI.stAudit_Ctrl.iBatchSelectedPhase)), STR2 := ': '), STR2 := GV.arrPhasesClean[GV.stActiveRecipe.stCleaning[GV.stHMI.stAudit_Ctrl.iBatchSelectedPhase].iType]), STR2 := ' - Phase 3 duration seconds'),
    iq_stParams := stDbParam,
    iq_bWrite := bWrite); // FB_AuditTrail_Write

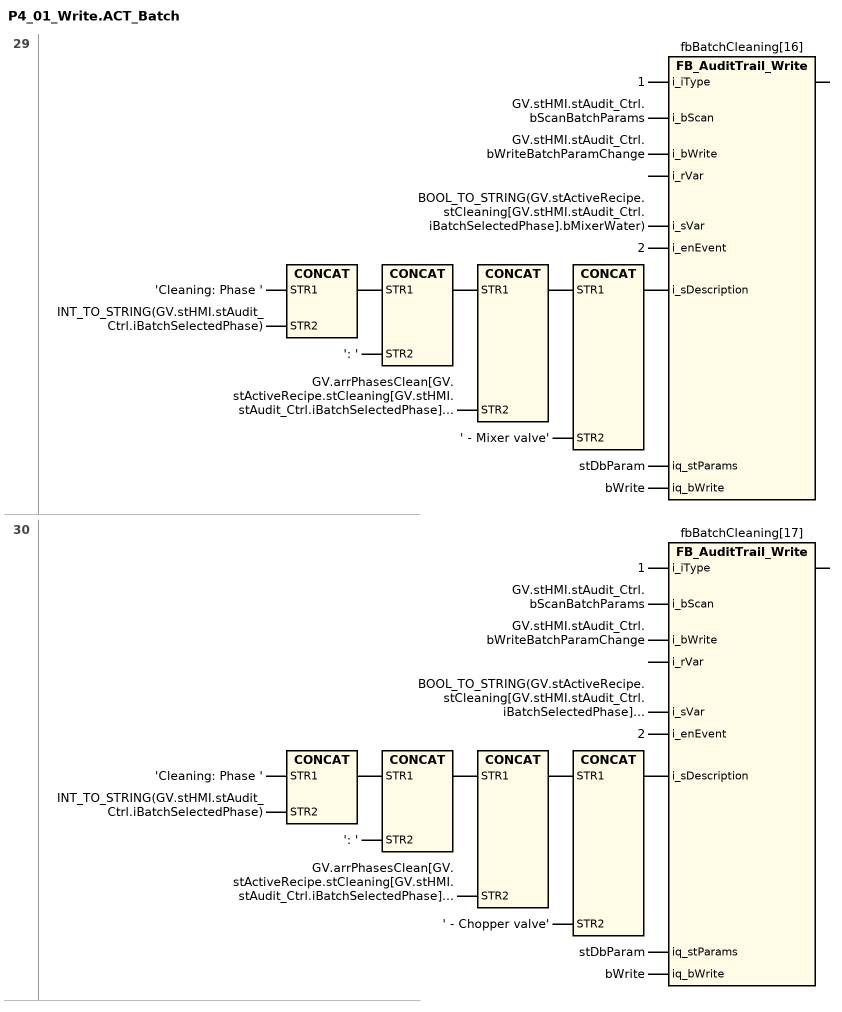
// NETWORK 29
fbBatchCleaning[16](
    i_iType := 1,
    i_bScan := GV.stHMI.stAudit_Ctrl.bScanBatchParams,
    i_bWrite := GV.stHMI.stAudit_Ctrl.bWriteBatchParamChange,
    i_sVar := BOOL_TO_STRING(GV.stActiveRecipe.stCleaning[GV.stHMI.stAudit_Ctrl.iBatchSelectedPhase].bMixerWater),
    i_enEvent := 2,
    i_sDescription := CONCAT(STR1 := CONCAT(STR1 := CONCAT(STR1 := CONCAT(STR1 := 'Cleaning: Phase ', STR2 := INT_TO_STRING(GV.stHMI.stAudit_Ctrl.iBatchSelectedPhase)), STR2 := ': '), STR2 := GV.arrPhasesClean[GV.stActiveRecipe.stCleaning[GV.stHMI.stAudit_Ctrl.iBatchSelectedPhase].iType]), STR2 := ' - Mixer valve'),
    iq_stParams := stDbParam,
    iq_bWrite := bWrite); // FB_AuditTrail_Write

// NETWORK 30
fbBatchCleaning[17](
    i_iType := 1,
    i_bScan := GV.stHMI.stAudit_Ctrl.bScanBatchParams,
    i_bWrite := GV.stHMI.stAudit_Ctrl.bWriteBatchParamChange,
    i_sVar := BOOL_TO_STRING(GV.stActiveRecipe.stCleaning[GV.stHMI.stAudit_Ctrl.iBatchSelectedPhase].bChopperWater),
    i_enEvent := 2,
    i_sDescription := CONCAT(STR1 := CONCAT(STR1 := CONCAT(STR1 := CONCAT(STR1 := 'Cleaning: Phase ', STR2 := INT_TO_STRING(GV.stHMI.stAudit_Ctrl.iBatchSelectedPhase)), STR2 := ': '), STR2 := GV.arrPhasesClean[GV.stActiveRecipe.stCleaning[GV.stHMI.stAudit_Ctrl.iBatchSelectedPhase].iType]), STR2 := ' - Chopper valve'),
    iq_stParams := stDbParam,
    iq_bWrite := bWrite); // FB_AuditTrail_Write

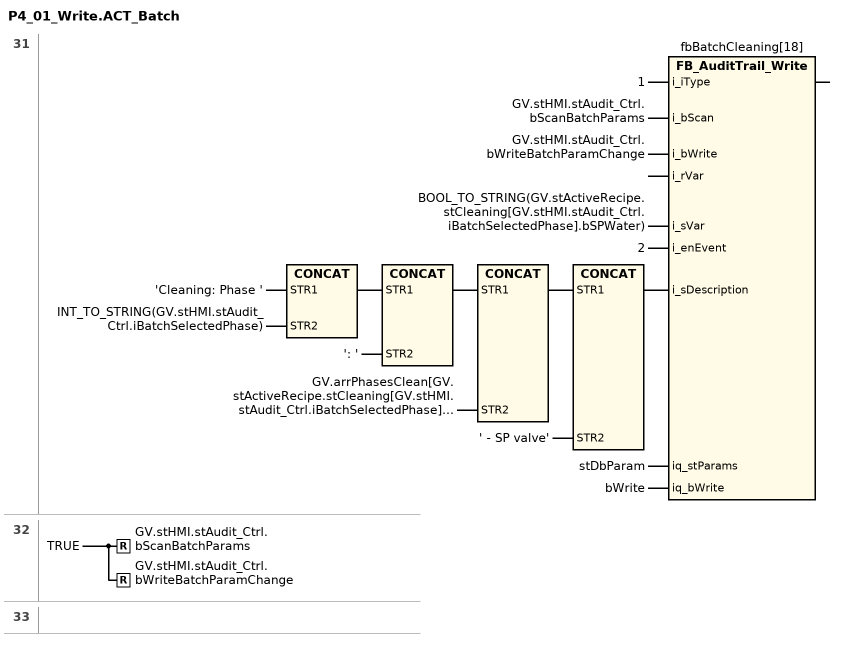
// NETWORK 31
fbBatchCleaning[18](
    i_iType := 1,
    i_bScan := GV.stHMI.stAudit_Ctrl.bScanBatchParams,
    i_bWrite := GV.stHMI.stAudit_Ctrl.bWriteBatchParamChange,
    i_sVar := BOOL_TO_STRING(GV.stActiveRecipe.stCleaning[GV.stHMI.stAudit_Ctrl.iBatchSelectedPhase].bSPWater),
    i_enEvent := 2,
    i_sDescription := CONCAT(STR1 := CONCAT(STR1 := CONCAT(STR1 := CONCAT(STR1 := 'Cleaning: Phase ', STR2 := INT_TO_STRING(GV.stHMI.stAudit_Ctrl.iBatchSelectedPhase)), STR2 := ': '), STR2 := GV.arrPhasesClean[GV.stActiveRecipe.stCleaning[GV.stHMI.stAudit_Ctrl.iBatchSelectedPhase].iType]), STR2 := ' - SP valve'),
    iq_stParams := stDbParam,
    iq_bWrite := bWrite); // FB_AuditTrail_Write

// NETWORK 32
GV.stHMI.stAudit_Ctrl.bScanBatchParams R= TRUE;
GV.stHMI.stAudit_Ctrl.bWriteBatchParamChange R= TRUE;

// NETWORK 33
END_ACTION

ACTION ACT_General:
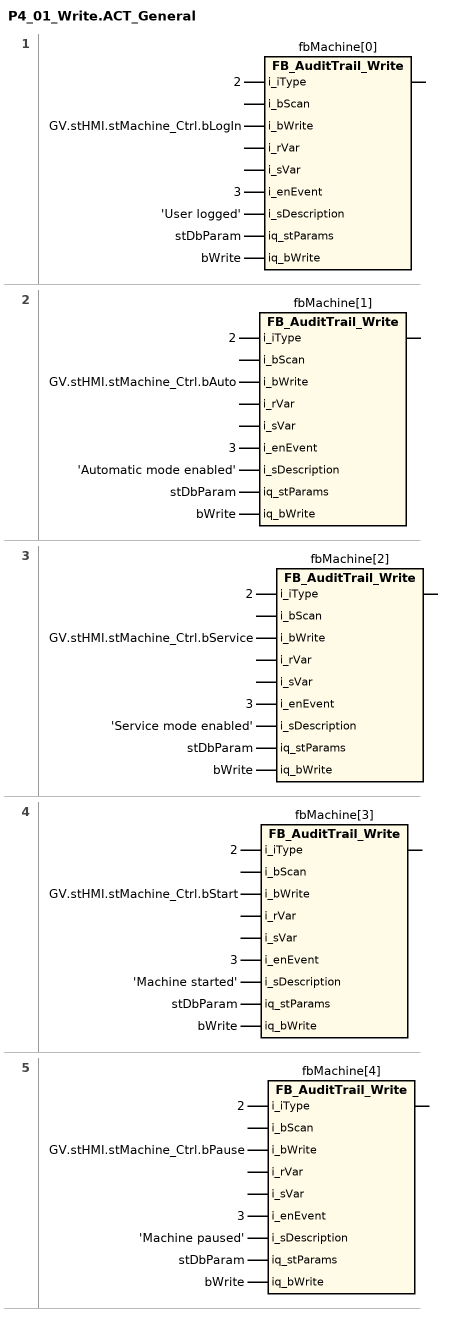
// NETWORK 1
fbMachine[0](
    i_iType := 2,
    i_bWrite := GV.stHMI.stMachine_Ctrl.bLogIn,
    i_enEvent := 3,
    i_sDescription := 'User logged',
    iq_stParams := stDbParam,
    iq_bWrite := bWrite); // FB_AuditTrail_Write

// NETWORK 2
fbMachine[1](
    i_iType := 2,
    i_bWrite := GV.stHMI.stMachine_Ctrl.bAuto,
    i_enEvent := 3,
    i_sDescription := 'Automatic mode enabled',
    iq_stParams := stDbParam,
    iq_bWrite := bWrite); // FB_AuditTrail_Write

// NETWORK 3
fbMachine[2](
    i_iType := 2,
    i_bWrite := GV.stHMI.stMachine_Ctrl.bService,
    i_enEvent := 3,
    i_sDescription := 'Service mode enabled',
    iq_stParams := stDbParam,
    iq_bWrite := bWrite); // FB_AuditTrail_Write

// NETWORK 4
fbMachine[3](
    i_iType := 2,
    i_bWrite := GV.stHMI.stMachine_Ctrl.bStart,
    i_enEvent := 3,
    i_sDescription := 'Machine started',
    iq_stParams := stDbParam,
    iq_bWrite := bWrite); // FB_AuditTrail_Write

// NETWORK 5
fbMachine[4](
    i_iType := 2,
    i_bWrite := GV.stHMI.stMachine_Ctrl.bPause,
    i_enEvent := 3,
    i_sDescription := 'Machine paused',
    iq_stParams := stDbParam,
    iq_bWrite := bWrite); // FB_AuditTrail_Write

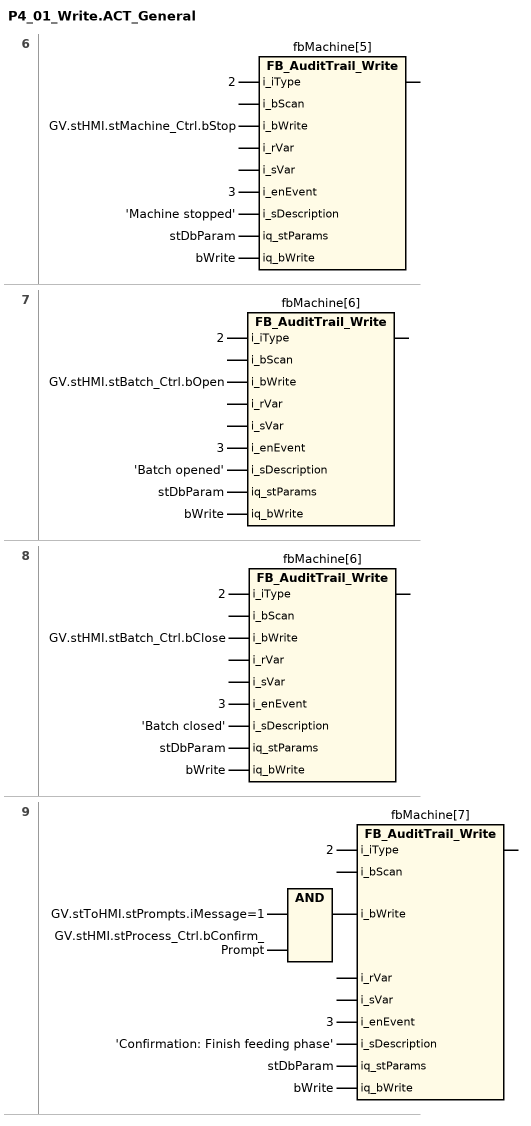
// NETWORK 6
fbMachine[5](
    i_iType := 2,
    i_bWrite := GV.stHMI.stMachine_Ctrl.bStop,
    i_enEvent := 3,
    i_sDescription := 'Machine stopped',
    iq_stParams := stDbParam,
    iq_bWrite := bWrite); // FB_AuditTrail_Write

// NETWORK 7
fbMachine[6](
    i_iType := 2,
    i_bWrite := GV.stHMI.stBatch_Ctrl.bOpen,
    i_enEvent := 3,
    i_sDescription := 'Batch opened',
    iq_stParams := stDbParam,
    iq_bWrite := bWrite); // FB_AuditTrail_Write

// NETWORK 8
fbMachine[6](
    i_iType := 2,
    i_bWrite := GV.stHMI.stBatch_Ctrl.bClose,
    i_enEvent := 3,
    i_sDescription := 'Batch closed',
    iq_stParams := stDbParam,
    iq_bWrite := bWrite); // FB_AuditTrail_Write

// NETWORK 9
fbMachine[7](
    i_iType := 2,
    i_bWrite := (GV.stToHMI.stPrompts.iMessage=1) AND GV.stHMI.stProcess_Ctrl.bConfirm_Prompt,
    i_enEvent := 3,
    i_sDescription := 'Confirmation: Finish feeding phase',
    iq_stParams := stDbParam,
    iq_bWrite := bWrite); // FB_AuditTrail_Write

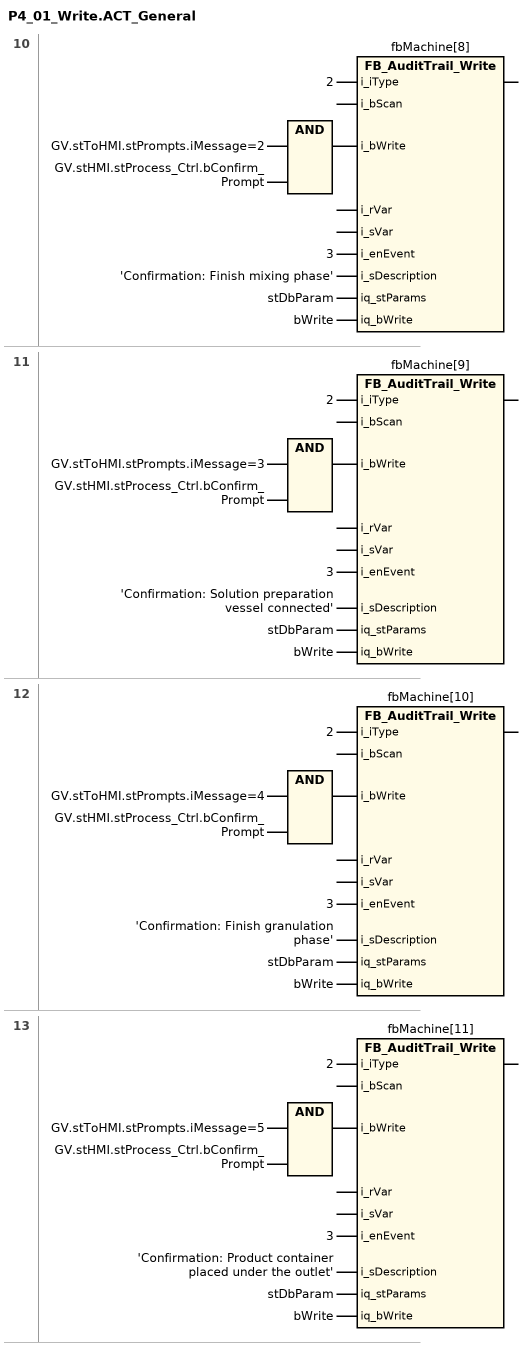
// NETWORK 10
fbMachine[8](
    i_iType := 2,
    i_bWrite := (GV.stToHMI.stPrompts.iMessage=2) AND GV.stHMI.stProcess_Ctrl.bConfirm_Prompt,
    i_enEvent := 3,
    i_sDescription := 'Confirmation: Finish mixing phase',
    iq_stParams := stDbParam,
    iq_bWrite := bWrite); // FB_AuditTrail_Write

// NETWORK 11
fbMachine[9](
    i_iType := 2,
    i_bWrite := (GV.stToHMI.stPrompts.iMessage=3) AND GV.stHMI.stProcess_Ctrl.bConfirm_Prompt,
    i_enEvent := 3,
    i_sDescription := 'Confirmation: Solution preparation vessel connected',
    iq_stParams := stDbParam,
    iq_bWrite := bWrite); // FB_AuditTrail_Write

// NETWORK 12
fbMachine[10](
    i_iType := 2,
    i_bWrite := (GV.stToHMI.stPrompts.iMessage=4) AND GV.stHMI.stProcess_Ctrl.bConfirm_Prompt,
    i_enEvent := 3,
    i_sDescription := 'Confirmation: Finish granulation phase',
    iq_stParams := stDbParam,
    iq_bWrite := bWrite); // FB_AuditTrail_Write

// NETWORK 13
fbMachine[11](
    i_iType := 2,
    i_bWrite := (GV.stToHMI.stPrompts.iMessage=5) AND GV.stHMI.stProcess_Ctrl.bConfirm_Prompt,
    i_enEvent := 3,
    i_sDescription := 'Confirmation: Product container placed under the outlet',
    iq_stParams := stDbParam,
    iq_bWrite := bWrite); // FB_AuditTrail_Write

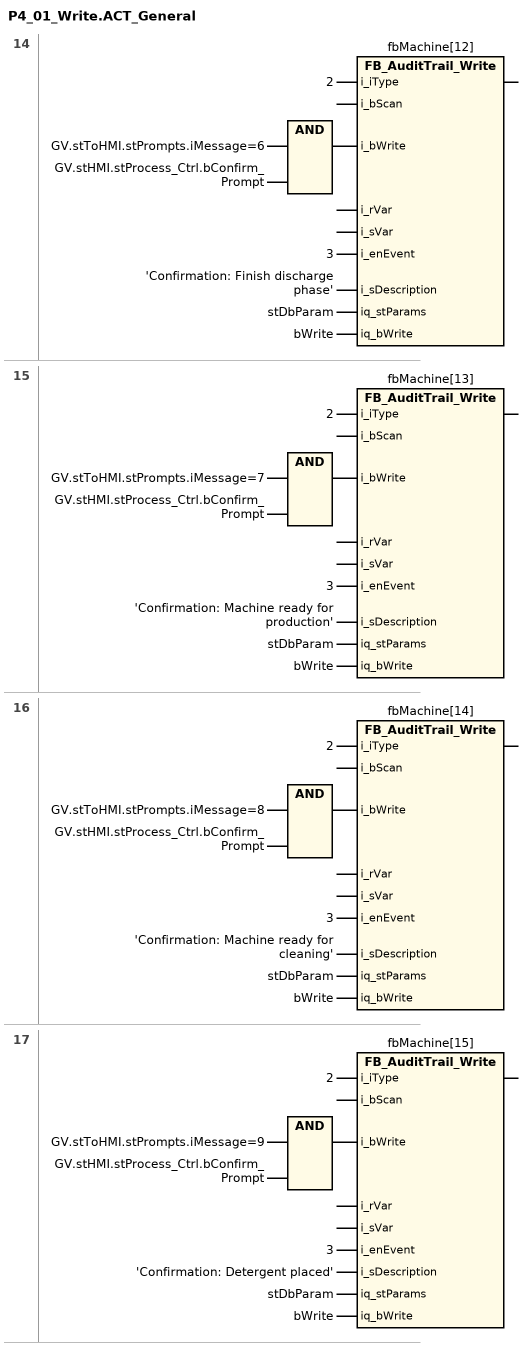
// NETWORK 14
fbMachine[12](
    i_iType := 2,
    i_bWrite := (GV.stToHMI.stPrompts.iMessage=6) AND GV.stHMI.stProcess_Ctrl.bConfirm_Prompt,
    i_enEvent := 3,
    i_sDescription := 'Confirmation: Finish discharge phase',
    iq_stParams := stDbParam,
    iq_bWrite := bWrite); // FB_AuditTrail_Write

// NETWORK 15
fbMachine[13](
    i_iType := 2,
    i_bWrite := (GV.stToHMI.stPrompts.iMessage=7) AND GV.stHMI.stProcess_Ctrl.bConfirm_Prompt,
    i_enEvent := 3,
    i_sDescription := 'Confirmation: Machine ready for production',
    iq_stParams := stDbParam,
    iq_bWrite := bWrite); // FB_AuditTrail_Write

// NETWORK 16
fbMachine[14](
    i_iType := 2,
    i_bWrite := (GV.stToHMI.stPrompts.iMessage=8) AND GV.stHMI.stProcess_Ctrl.bConfirm_Prompt,
    i_enEvent := 3,
    i_sDescription := 'Confirmation: Machine ready for cleaning',
    iq_stParams := stDbParam,
    iq_bWrite := bWrite); // FB_AuditTrail_Write

// NETWORK 17
fbMachine[15](
    i_iType := 2,
    i_bWrite := (GV.stToHMI.stPrompts.iMessage=9) AND GV.stHMI.stProcess_Ctrl.bConfirm_Prompt,
    i_enEvent := 3,
    i_sDescription := 'Confirmation: Detergent placed',
    iq_stParams := stDbParam,
    iq_bWrite := bWrite); // FB_AuditTrail_Write

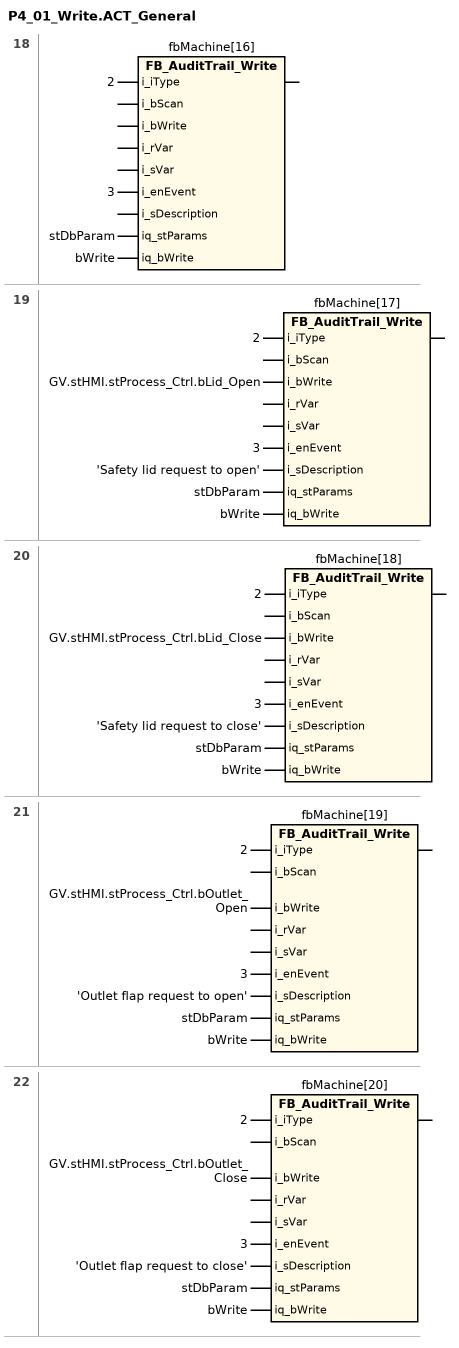
// NETWORK 18
fbMachine[16](i_iType := 2, i_enEvent := 3, iq_stParams := stDbParam, iq_bWrite := bWrite); // FB_AuditTrail_Write

// NETWORK 19
fbMachine[17](
    i_iType := 2,
    i_bWrite := GV.stHMI.stProcess_Ctrl.bLid_Open,
    i_enEvent := 3,
    i_sDescription := 'Safety lid request to open',
    iq_stParams := stDbParam,
    iq_bWrite := bWrite); // FB_AuditTrail_Write

// NETWORK 20
fbMachine[18](
    i_iType := 2,
    i_bWrite := GV.stHMI.stProcess_Ctrl.bLid_Close,
    i_enEvent := 3,
    i_sDescription := 'Safety lid request to close',
    iq_stParams := stDbParam,
    iq_bWrite := bWrite); // FB_AuditTrail_Write

// NETWORK 21
fbMachine[19](
    i_iType := 2,
    i_bWrite := GV.stHMI.stProcess_Ctrl.bOutlet_Open,
    i_enEvent := 3,
    i_sDescription := 'Outlet flap request to open',
    iq_stParams := stDbParam,
    iq_bWrite := bWrite); // FB_AuditTrail_Write

// NETWORK 22
fbMachine[20](
    i_iType := 2,
    i_bWrite := GV.stHMI.stProcess_Ctrl.bOutlet_Close,
    i_enEvent := 3,
    i_sDescription := 'Outlet flap request to close',
    iq_stParams := stDbParam,
    iq_bWrite := bWrite); // FB_AuditTrail_Write

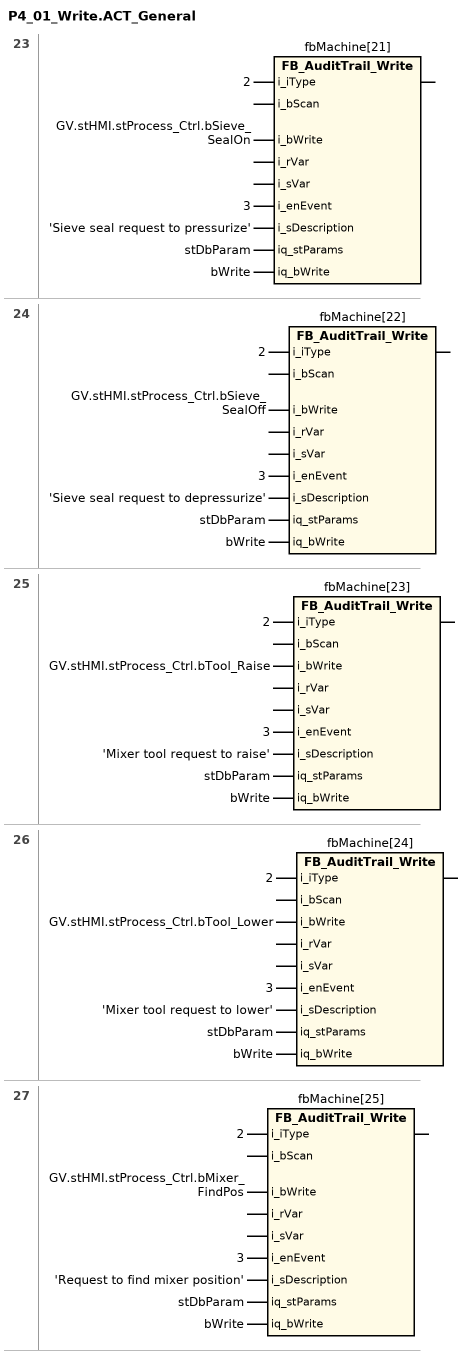
// NETWORK 23
fbMachine[21](
    i_iType := 2,
    i_bWrite := GV.stHMI.stProcess_Ctrl.bSieve_SealOn,
    i_enEvent := 3,
    i_sDescription := 'Sieve seal request to pressurize',
    iq_stParams := stDbParam,
    iq_bWrite := bWrite); // FB_AuditTrail_Write

// NETWORK 24
fbMachine[22](
    i_iType := 2,
    i_bWrite := GV.stHMI.stProcess_Ctrl.bSieve_SealOff,
    i_enEvent := 3,
    i_sDescription := 'Sieve seal request to depressurize',
    iq_stParams := stDbParam,
    iq_bWrite := bWrite); // FB_AuditTrail_Write

// NETWORK 25
fbMachine[23](
    i_iType := 2,
    i_bWrite := GV.stHMI.stProcess_Ctrl.bTool_Raise,
    i_enEvent := 3,
    i_sDescription := 'Mixer tool request to raise',
    iq_stParams := stDbParam,
    iq_bWrite := bWrite); // FB_AuditTrail_Write

// NETWORK 26
fbMachine[24](
    i_iType := 2,
    i_bWrite := GV.stHMI.stProcess_Ctrl.bTool_Lower,
    i_enEvent := 3,
    i_sDescription := 'Mixer tool request to lower',
    iq_stParams := stDbParam,
    iq_bWrite := bWrite); // FB_AuditTrail_Write

// NETWORK 27
fbMachine[25](
    i_iType := 2,
    i_bWrite := GV.stHMI.stProcess_Ctrl.bMixer_FindPos,
    i_enEvent := 3,
    i_sDescription := 'Request to find mixer position',
    iq_stParams := stDbParam,
    iq_bWrite := bWrite); // FB_AuditTrail_Write

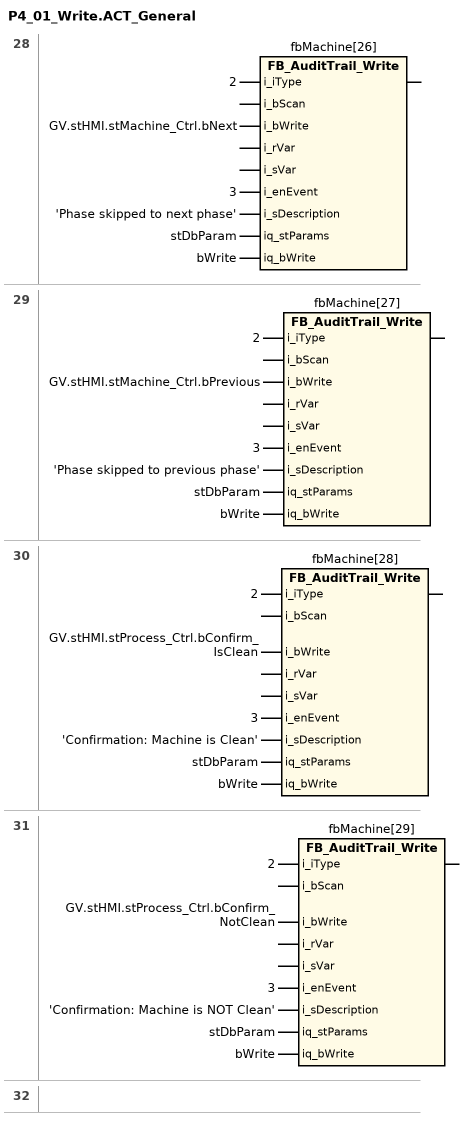
// NETWORK 28
fbMachine[26](
    i_iType := 2,
    i_bWrite := GV.stHMI.stMachine_Ctrl.bNext,
    i_enEvent := 3,
    i_sDescription := 'Phase skipped to next phase',
    iq_stParams := stDbParam,
    iq_bWrite := bWrite); // FB_AuditTrail_Write

// NETWORK 29
fbMachine[27](
    i_iType := 2,
    i_bWrite := GV.stHMI.stMachine_Ctrl.bPrevious,
    i_enEvent := 3,
    i_sDescription := 'Phase skipped to previous phase',
    iq_stParams := stDbParam,
    iq_bWrite := bWrite); // FB_AuditTrail_Write

// NETWORK 30
fbMachine[28](
    i_iType := 2,
    i_bWrite := GV.stHMI.stProcess_Ctrl.bConfirm_IsClean,
    i_enEvent := 3,
    i_sDescription := 'Confirmation: Machine is Clean',
    iq_stParams := stDbParam,
    iq_bWrite := bWrite); // FB_AuditTrail_Write

// NETWORK 31
fbMachine[29](
    i_iType := 2,
    i_bWrite := GV.stHMI.stProcess_Ctrl.bConfirm_NotClean,
    i_enEvent := 3,
    i_sDescription := 'Confirmation: Machine is NOT Clean',
    iq_stParams := stDbParam,
    iq_bWrite := bWrite); // FB_AuditTrail_Write

// NETWORK 32
END_ACTION

ACTION ACT_Recipe:
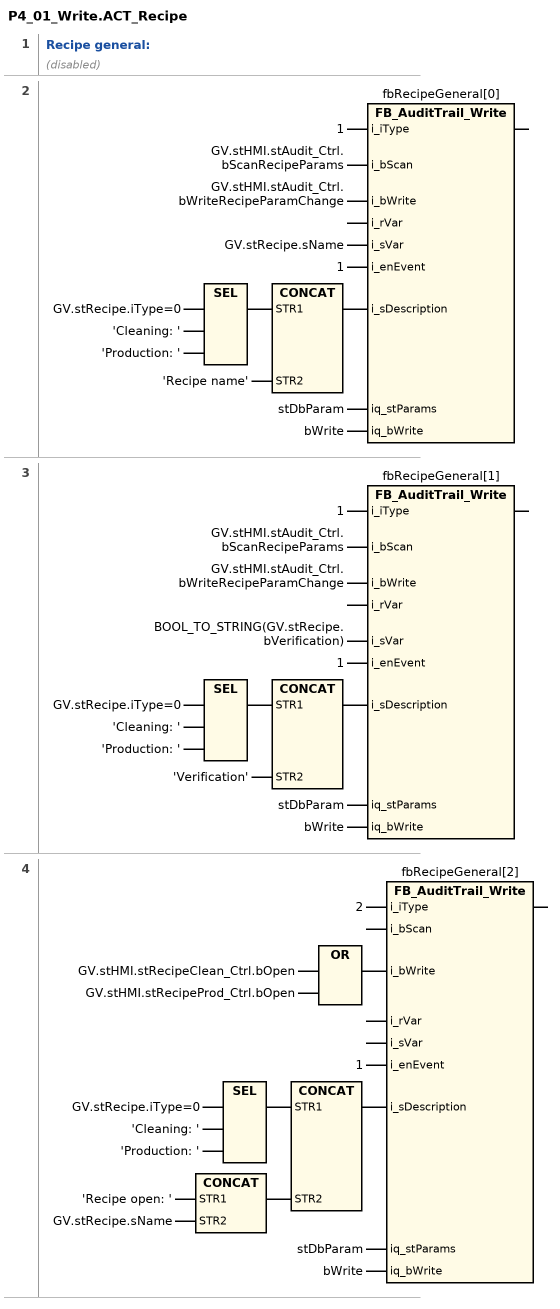
// NETWORK 1 (disabled)
// label: Recipe general

// NETWORK 2
fbRecipeGeneral[0](
    i_iType := 1,
    i_bScan := GV.stHMI.stAudit_Ctrl.bScanRecipeParams,
    i_bWrite := GV.stHMI.stAudit_Ctrl.bWriteRecipeParamChange,
    i_sVar := GV.stRecipe.sName,
    i_enEvent := 1,
    i_sDescription := CONCAT(STR1 := SEL(GV.stRecipe.iType=0, 'Cleaning: ', 'Production: '), STR2 := 'Recipe name'),
    iq_stParams := stDbParam,
    iq_bWrite := bWrite); // FB_AuditTrail_Write

// NETWORK 3
fbRecipeGeneral[1](
    i_iType := 1,
    i_bScan := GV.stHMI.stAudit_Ctrl.bScanRecipeParams,
    i_bWrite := GV.stHMI.stAudit_Ctrl.bWriteRecipeParamChange,
    i_sVar := BOOL_TO_STRING(GV.stRecipe.bVerification),
    i_enEvent := 1,
    i_sDescription := CONCAT(STR1 := SEL(GV.stRecipe.iType=0, 'Cleaning: ', 'Production: '), STR2 := 'Verification'),
    iq_stParams := stDbParam,
    iq_bWrite := bWrite); // FB_AuditTrail_Write

// NETWORK 4
fbRecipeGeneral[2](
    i_iType := 2,
    i_bWrite := GV.stHMI.stRecipeClean_Ctrl.bOpen OR GV.stHMI.stRecipeProd_Ctrl.bOpen,
    i_enEvent := 1,
    i_sDescription := CONCAT(STR1 := SEL(GV.stRecipe.iType=0, 'Cleaning: ', 'Production: '), STR2 := CONCAT(STR1 := 'Recipe open: ', STR2 := GV.stRecipe.sName)),
    iq_stParams := stDbParam,
    iq_bWrite := bWrite); // FB_AuditTrail_Write

